// TwinCAT 3 PLC project Sample01
// ProgramVersion: 3.1.4020.10
// libraries:
//   Tc2_Standard, * (Beckhoff Automation GmbH)
//   Tc2_System, * (Beckhoff Automation GmbH)
//   Tc3_Module, * (Beckhoff Automation GmbH)
// project tree:
//   DUTs/ E_LampType.TcDUT
//   / PlcTask.TcTTO (not stored)
//   POUs/ Class Diagram.TcCD (not stored), FB_AnalogValue.TcPOU, FB_Controller.TcPOU, FB_LampUpDown.TcPOU, FB_LampSetDirect.TcPOU, FB_LampOnOff.TcPOU, I_Observer.TcIO, I_Subject.TcIO, MAIN.TcPOU
// real-time tasks:
//   TASK PlcTask: cycle T#10ms, priority 20, ADS port 350

// ---- DUTs/E_LampType.TcDUT
{attribute 'qualified_only'}
{attribute 'strict'}
TYPE E_LampType :
(
	Unknown := -1,
	SetDirect := 0,
	OnOff := 1,
	UpDown := 2
) := Unknown;
END_TYPE

// ---- POUs/I_Observer.TcIO
INTERFACE I_Observer

METHOD Update : BYTE
VAR_INPUT
	nNewValue		:	BYTE(0..100);
END_VAR
END_METHOD

END_INTERFACE

// ---- POUs/I_Subject.TcIO
INTERFACE I_Subject

METHOD Attach
VAR_INPUT
	ipObserver	: I_Observer;
END_VAR
END_METHOD

METHOD Detach
VAR_INPUT
END_VAR
END_METHOD

END_INTERFACE

// ---- POUs/FB_AnalogValue.TcPOU
FUNCTION_BLOCK PUBLIC FB_AnalogValue IMPLEMENTS I_Observer
VAR
	_nActualValue		:	BYTE(0..100);
END_VAR

PROPERTY nValue : BYTE (0..100)
GET
nValue := _nActualValue;
END_GET
END_PROPERTY

METHOD Update : BYTE
VAR_INPUT
	nNewValue		:	BYTE(0..100);
END_VAR
_nActualValue := nNewValue;
END_METHOD

END_FUNCTION_BLOCK

// ---- POUs/FB_Controller.TcPOU
FUNCTION_BLOCK PUBLIC FB_Controller
VAR
	fbLampOnOff			:	FB_LampOnOff();
	fbLampSetDirect		:	FB_LampSetDirect();
	fbLampUpDown		:	FB_LampUpDown();
	fbActualValue		:	FB_AnalogValue();
	_eActiveLamp		:	E_LampType;
END_VAR

// Reduces the control value by 5 in the range of 10 to 100. 
METHOD PUBLIC DimDown
CASE _eActiveLamp OF
	E_LampType.OnOff:
		fbLampOnOff.Off();
	E_LampType.SetDirect:
		IF (fbActualValue.nValue >= 15) THEN
			fbLampSetDirect.SetLightLevel(fbActualValue.nValue - 5);
		END_IF
	E_LampType.UpDown:
		IF (fbActualValue.nValue >= 15) THEN
			fbLampUpDown.OneStepDown();
			fbLampUpDown.OneStepDown();
			fbLampUpDown.OneStepDown();
			fbLampUpDown.OneStepDown();
			fbLampUpDown.OneStepDown();
		END_IF
END_CASE
END_METHOD

// Increments the control value by 5 in the range of 10 to 100.
METHOD PUBLIC DimUp
CASE _eActiveLamp OF
	E_LampType.OnOff:
		fbLampOnOff.On();
	E_LampType.SetDirect:
		IF (fbActualValue.nValue <= 95) THEN
			fbLampSetDirect.SetLightLevel(fbActualValue.nValue + 5);
		END_IF
	E_LampType.UpDown:
		IF (fbActualValue.nValue <= 95) THEN
			fbLampUpDown.OneStepUp();
			fbLampUpDown.OneStepUp();
			fbLampUpDown.OneStepUp();
			fbLampUpDown.OneStepUp();
			fbLampUpDown.OneStepUp();
		END_IF
END_CASE
END_METHOD

{attribute 'monitoring' := 'variable'}
PROPERTY PUBLIC eActiveLamp : E_LampType
GET
eActiveLamp := _eActiveLamp;
END_GET
SET
Off();

fbLampOnOff.Detach();
fbLampSetDirect.Detach();
fbLampUpDown.Detach();

CASE eActiveLamp OF
	E_LampType.OnOff:
		fbLampOnOff.Attach(fbActualValue);
	E_LampType.SetDirect:
		fbLampSetDirect.Attach(fbActualValue);
	E_LampType.UpDown:
		fbLampUpDown.Attach(fbActualValue);
END_CASE

_eActiveLamp := eActiveLamp;
END_SET
END_PROPERTY

// Sets the control value to 0.
METHOD PUBLIC Off
CASE _eActiveLamp OF
	E_LampType.OnOff:
		fbLampOnOff.Off();
	E_LampType.SetDirect:
		fbLampSetDirect.SetLightLevel(0);
	E_LampType.UpDown:
		IF (fbActualValue.nValue > 0) THEN
			fbLampUpDown.OnOff();
		END_IF
END_CASE
END_METHOD

// Sets the control value to 100.
METHOD PUBLIC On
CASE _eActiveLamp OF
	E_LampType.OnOff:
		fbLampOnOff.On();
	E_LampType.SetDirect:
		fbLampSetDirect.SetLightLevel(100);
	E_LampType.UpDown:
		IF (fbActualValue.nValue = 0) THEN
			fbLampUpDown.OnOff();
		END_IF
END_CASE
END_METHOD

END_FUNCTION_BLOCK

// ---- POUs/FB_LampOnOff.TcPOU
FUNCTION_BLOCK PUBLIC FB_LampOnOff IMPLEMENTS I_Subject
VAR
	nLightLevel			:	BYTE(0..100);
	_ipObserver			:	I_Observer;	
END_VAR

METHOD Attach
VAR_INPUT
	ipObserver		: I_Observer;
END_VAR
IF (ipObserver = 0) THEN
	RETURN;
END_IF
_ipObserver := ipObserver;
END_METHOD

METHOD Detach
_ipObserver := 0;
END_METHOD

// Sets the control value to 0.
METHOD PUBLIC Off
nLightLevel := 0;
IF (_ipObserver <> 0) THEN
	_ipObserver.Update(nLightLevel);
END_IF
END_METHOD

// Sets the control value to 100.
METHOD PUBLIC On
nLightLevel := 100;
IF (_ipObserver <> 0) THEN
	_ipObserver.Update(nLightLevel);
END_IF
END_METHOD

END_FUNCTION_BLOCK

// ---- POUs/FB_LampSetDirect.TcPOU
FUNCTION_BLOCK PUBLIC FB_LampSetDirect IMPLEMENTS I_Subject
VAR
	nLightLevel			:	BYTE(0..100);
	_ipObserver			:	I_Observer;	
END_VAR

METHOD Attach
VAR_INPUT
	ipObserver		: I_Observer;
END_VAR
IF (ipObserver = 0) THEN
	RETURN;
END_IF
_ipObserver := ipObserver;
END_METHOD

METHOD Detach
_ipObserver := 0;
END_METHOD

// Sets the control value to a value between 0 and 100.
METHOD PUBLIC SetLightLevel
VAR_INPUT
	nNewLightLevel		:	BYTE(0..100);
END_VAR
nLightLevel := nNewLightLevel;
IF (_ipObserver <> 0) THEN
	_ipObserver.Update(nLightLevel);
END_IF
END_METHOD

END_FUNCTION_BLOCK

// ---- POUs/FB_LampUpDown.TcPOU
FUNCTION_BLOCK FB_LampUpDown IMPLEMENTS I_Subject
VAR
	nLightLevel			:	BYTE(0..100);
	_ipObserver			:	I_Observer;	
END_VAR

METHOD Attach
VAR_INPUT
	ipObserver		: I_Observer;
END_VAR
IF (ipObserver = 0) THEN
	RETURN;
END_IF
_ipObserver := ipObserver;
END_METHOD

METHOD Detach
_ipObserver := 0;
END_METHOD

// Reduces the control value by 1 in the range of 10 to 100. 
METHOD PUBLIC OneStepDown
nLightLevel := nLightLevel - 1;
IF (nLightLevel < 10) THEN
	nLightLevel := 10;
END_IF
IF (_ipObserver <> 0) THEN
	_ipObserver.Update(nLightLevel);
END_IF
END_METHOD

// Increments the control value by 1 in the range of 10 to 100.
METHOD PUBLIC OneStepUp
nLightLevel := nLightLevel + 1;
IF (nLightLevel > 100) THEN
	nLightLevel := 100;
END_IF
IF (_ipObserver <> 0) THEN
	_ipObserver.Update(nLightLevel);
END_IF
END_METHOD

// Toggles the control value between 0 and 100.
METHOD PUBLIC OnOff
IF (nLightLevel > 0) THEN
	nLightLevel := 0;
ELSE
	nLightLevel := 100;
END_IF
IF (_ipObserver <> 0) THEN
	_ipObserver.Update(nLightLevel);
end_IF
END_METHOD

END_FUNCTION_BLOCK

// ---- POUs/MAIN.TcPOU
PROGRAM MAIN
VAR
	fbController		:	FB_Controller();
	eActiveLamp 		:	E_LampType;
	bSetActiveLamp 		:	BOOL;
	bDimUp, bDimDown	:	BOOL;
	bOff, bOn			:	BOOL;
END_VAR

IF (bSetActiveLamp) THEN
	fbController.eActiveLamp := eActiveLamp;
	bSetActiveLamp := FALSE;
END_IF

IF (bDimUp) THEN
	fbController.DimUp();
	bDimUp := FALSE;
END_IF

IF (bDimDown) THEN
	fbController.DimDown();
	bDimDown := FALSE;
END_IF

IF (bOff) THEN
	fbController.Off();
	bOff := FALSE;
END_IF

IF (bOn) THEN
	fbController.On();
	bOn := FALSE;
END_IF

END_PROGRAM
